# EPICS substitutions: Db/vac_ctrl_tpg300.substitutions
file vac_ctrl_tpg300_common.template
{
	pattern { NULL }

		{ "" }
}

file vac_ctrl_tpg300_sensor.template
{
	pattern { SENSOR,  SLOT,  SOURCE }

		{ A1,      A,     A }
		{ A2,      A,     B }
		{ B1,      B,     C }
		{ B2,      B,     D }
}

file vac_ctrl_tpg300_relay.template
{
	pattern { FUNCTION }

		{ 1 }
		{ 2 }
		{ 3 }
		{ 4 }
}
